FUNCTION_BLOCK CylControlIL (* Basic Function Block Type *)
  (* Standard: 61499-2 *)
  (* Version 0.0, 11/30/2015, paarnio, nxtControl GmbH, Template *)
  PACKAGE Main;
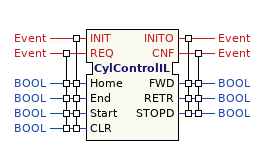
  EVENT_INPUT
    INIT WITH Home, End, Start, CLR; (* Initialization Request *)
    REQ WITH Home, End, Start, CLR; (* Normal Execution Request *)
  END_EVENT
  EVENT_OUTPUT
    INITO WITH FWD, RETR, STOPD; (* Initialization Confirm *)
    CNF WITH FWD, RETR, STOPD; (* Execution Confirmation *)
  END_EVENT
  VAR_INPUT
    Home : BOOL;
    End : BOOL;
    Start : BOOL;
    CLR : BOOL;
  END_VAR
  VAR_OUTPUT
    FWD : BOOL;
    RETR : BOOL;
    STOPD : BOOL;
  END_VAR
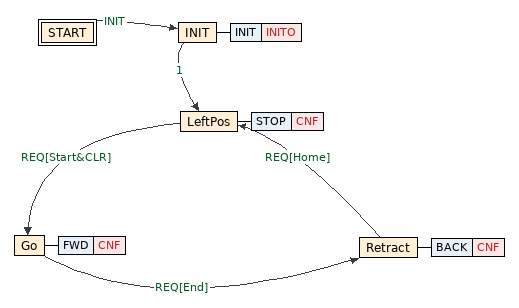
  EC_STATES
    START; (* Initial State *)
    INIT : INIT -> INITO; (* Initialization *)
    Go : FWD -> CNF;
    Retract : BACK -> CNF;
    LeftPos : STOP -> CNF;
  END_STATES
  EC_TRANSITIONS
    START TO INIT := INIT;
    INIT TO LeftPos := 1;
    LeftPos TO Go := REQ[Start&CLR];
    Go TO Retract := REQ[End];
    Retract TO LeftPos := REQ[Home];
  END_TRANSITIONS
  ALGORITHM INIT IN ST: (* Initialization algorithm *)
FWD :=FALSE;
RETR:=FALSE;
STOPD:=TRUE;
//State:=0;
  END_ALGORITHM
  ALGORITHM FWD IN ST:
FWD :=TRUE;
STOPD:=FALSE;
//State:=2;
  END_ALGORITHM
  ALGORITHM BACK IN ST:
FWD :=FALSE;
RETR:=TRUE;
STOPD:=FALSE;
//State:=3;
  END_ALGORITHM
  ALGORITHM STOP IN ST:
FWD :=FALSE;
RETR:=FALSE;
STOPD:=TRUE;
//State:=1;
  END_ALGORITHM
END_FUNCTION_BLOCK
